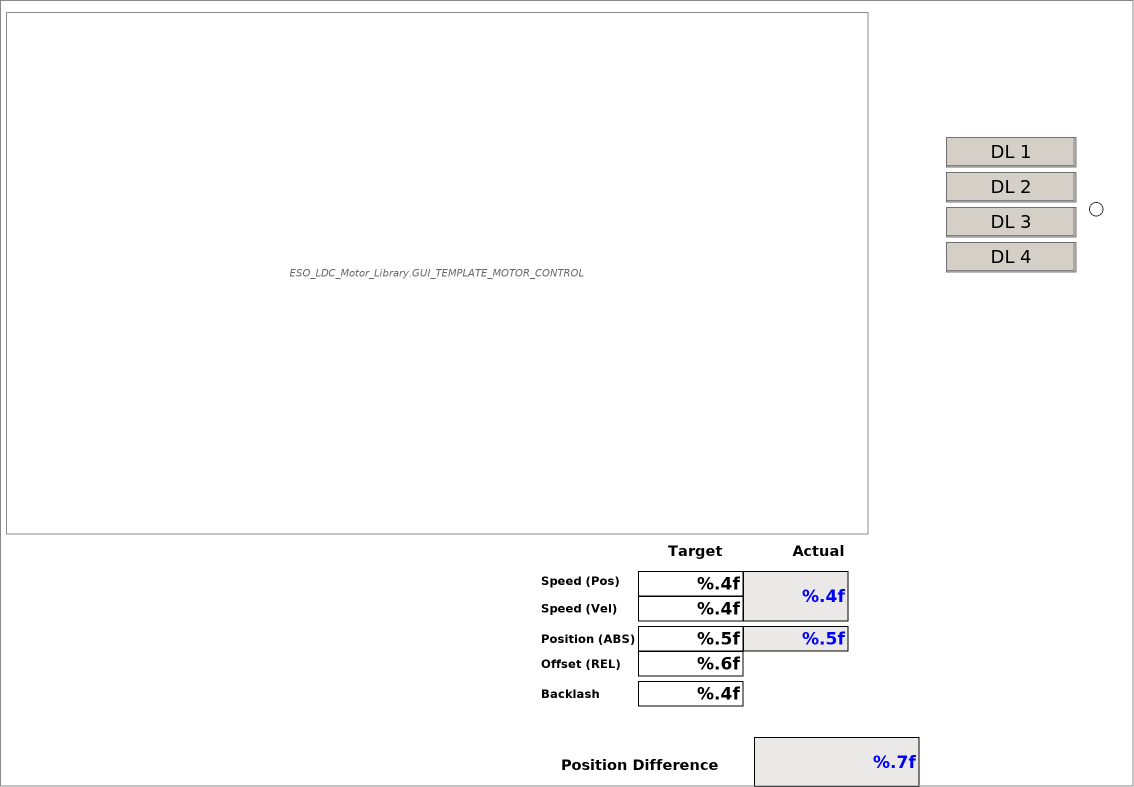
VISUALIZATION GUI_NOTT_DL_CTRL  // 1134x787
    RadioButton (1087,139 47x140), variable: MAIN.nott_ics.Delay_Lines.guiShutterIndex-1
        Areas[0]: Text=Radiobutton
        Areas[1]: Text=Radiobutton
    Button (946,137 130x30), "DL 1"
        OnMouseClick: execute { MAIN.nott_ics.Delay_Lines.guiShutterIndex := 1; }
    Button (946,172 130x30), "DL 2"
        OnMouseClick: execute { MAIN.nott_ics.Delay_Lines.guiShutterIndex := 2; }
    Button (946,207 130x30), "DL 3"
        OnMouseClick: execute { MAIN.nott_ics.Delay_Lines.guiShutterIndex := 3; }
    Button (946,242 130x30), "DL 4"
        OnMouseClick: execute { MAIN.nott_ics.Delay_Lines.guiShutterIndex := 4; }
    Frame (6,12 862x522)
        shows ESO_LDC_Motor_Library.GUI_TEMPLATE_MOTOR_CONTROL(m_Instance := MAIN.nott_ics.Delay_Lines.ptrDelayLines[MAIN.nott_ics.Delay_Lines.guiShutterIndex]^)
    Rectangle (538,571 95x20), "Speed (Pos)"
    Rectangle (743,626 105x25), "%.5f", text variable: MAIN.nott_ics.Delay_Lines.ptrDelayLines[MAIN.nott_ics.Delay_Lines.guiShutterIndex]^.stat.lrPosActual, input disabled if: false
    Rectangle (665,541 190x20), "Target Actual"
    Rectangle (538,629 95x20), "Position (ABS)"
    Rectangle (743,571 105x50), "%.4f", text variable: MAIN.nott_ics.Delay_Lines.ptrDelayLines[MAIN.nott_ics.Delay_Lines.guiShutterIndex]^.stat.lrVelActual, input disabled if: false
    Rectangle (638,596 105x25), "%.4f", text variable: MAIN.nott_ics.Delay_Lines.ptrDelayLines[MAIN.nott_ics.Delay_Lines.guiShutterIndex]^.ctrl.lrVelocity
        OnMouseDown: write the text variable via Default
    Rectangle (538,684 95x20), "Backlash"
    Rectangle (638,681 105x25), "%.4f", text variable: MAIN.nott_ics.Delay_Lines.ptrDelayLines[MAIN.nott_ics.Delay_Lines.guiShutterIndex]^.cfg.lrBacklash
        OnMouseDown: write the text variable via Default
    Rectangle (538,596 95x25), "Speed (Vel)"
    Rectangle (638,626 105x25), "%.5f", tooltip "Absolute position used by "MOVE ABS"", text variable: MAIN.nott_ics.Delay_Lines.ptrDelayLines[MAIN.nott_ics.Delay_Lines.guiShutterIndex]^.ctrl.lrPosition
        OnMouseDown: write the text variable via Default
    Rectangle (638,571 105x25), "%.4f", text variable: MAIN.nott_ics.Delay_Lines.ptrDelayLines[MAIN.nott_ics.Delay_Lines.guiShutterIndex]^.cfg.lrDefaultVelocity
        OnMouseDown: write the text variable via Default
    Rectangle (538,654 95x20), "Offset (REL)"
    Rectangle (638,651 105x25), "%.6f", tooltip "Relative offset used by "MOVE REL"", text variable: MAIN.nott_ics.Delay_Lines.ptrDelayLines[MAIN.nott_ics.Delay_Lines.guiShutterIndex]^.ctrl.lrOffset
        OnMouseDown: write the text variable via Default
    Rectangle (754,737 165x50), "%.7f", text variable: MAIN.nott_ics.Delay_Lines.ptrDelayLines[MAIN.nott_ics.Delay_Lines.guiShutterIndex]^.stat.lrPosError, input disabled if: false
    Rectangle (558,755 190x20), "Position Difference"
END_VISUALIZATION

(* stored: Version 1.1.0.1, ProductVersion 3.1.4024.12
   Visu GUI_NOTT_DL_CTRL: Id {c56b1069-9226-48d1-9840-ead84fe86c8a} *)
